FUNCTION_BLOCK FB_MockNciChannel EXTENDS FB_ComponentBase IMPLEMENTS I_NciChannel_GCode
VAR_INPUT
    MockIsGrouped      : BOOL;
    MockIsProgramLoaded: BOOL;
    MockIsReady        : BOOL;
    MockIsMoving       : BOOL;
    MockChannelError   : BOOL;
    MockChannelErrorId : UDINT;
END_VAR
VAR_OUTPUT
    BuildGroupCallCount : INT;
    LoadProgramCallCount: INT;
    StartCallCount      : INT;
    StopCallCount       : INT;
    UngroupCallCount    : INT;
    ResetCallCount      : INT;
    LoadedProgramPath   : STRING(255);
END_VAR

METHOD BuildGroup
BuildGroupCallCount := BuildGroupCallCount + 1;
END_METHOD

PROPERTY ChannelError : BOOL
GET
ChannelError := MockChannelError;
END_GET
END_PROPERTY

PROPERTY ChannelErrorId : UDINT
GET
ChannelErrorId := MockChannelErrorId;
END_GET
END_PROPERTY

PROPERTY IsGrouped : BOOL
GET
IsGrouped := MockIsGrouped;
END_GET
END_PROPERTY

PROPERTY IsMoving : BOOL
GET
IsMoving := MockIsMoving;
END_GET
END_PROPERTY

PROPERTY IsProgramLoaded : BOOL
GET
IsProgramLoaded := MockIsProgramLoaded;
END_GET
END_PROPERTY

PROPERTY IsReady : BOOL
GET
IsReady := MockIsReady;
END_GET
END_PROPERTY

METHOD LoadProgram
VAR_INPUT
    sProgramPath : STRING(255);
END_VAR
LoadProgramCallCount := LoadProgramCallCount + 1;
LoadedProgramPath := sProgramPath;
END_METHOD

METHOD ResetChannel
ResetCallCount := ResetCallCount + 1;
MockChannelError := FALSE;
MockChannelErrorId := 0;
END_METHOD

METHOD Start
StartCallCount := StartCallCount + 1;
END_METHOD

METHOD Stop
StopCallCount := StopCallCount + 1;
END_METHOD

METHOD Ungroup
UngroupCallCount := UngroupCallCount + 1;
END_METHOD

END_FUNCTION_BLOCK

(* stored: Version 1.1.0.1, ProductVersion 3.1.4024.15
   POU FB_MockNciChannel: Id {c1b2c3d4-e5f6-4789-9999-000000000010}, SpecialFunc None
   Method BuildGroup: Id {a1b2c3d4-e5f6-4789-9999-000000000011}
   Property ChannelError: Id {a1b2c3d4-e5f6-4789-9999-000000000012}
   Get Get: Id {a1b2c3d4-e5f6-4789-9999-000000000013}
   Property ChannelErrorId: Id {a1b2c3d4-e5f6-4789-9999-000000000014}
   Get Get: Id {a1b2c3d4-e5f6-4789-9999-000000000015}
   Property IsGrouped: Id {a1b2c3d4-e5f6-4789-9999-000000000016}
   Get Get: Id {a1b2c3d4-e5f6-4789-9999-000000000017}
   Property IsMoving: Id {a1b2c3d4-e5f6-4789-9999-000000000018}
   Get Get: Id {a1b2c3d4-e5f6-4789-9999-000000000019}
   Property IsProgramLoaded: Id {a1b2c3d4-e5f6-4789-9999-000000000020}
   Get Get: Id {a1b2c3d4-e5f6-4789-9999-000000000021}
   Property IsReady: Id {a1b2c3d4-e5f6-4789-9999-000000000022}
   Get Get: Id {a1b2c3d4-e5f6-4789-9999-000000000023}
   Method LoadProgram: Id {a1b2c3d4-e5f6-4789-9999-000000000024}
   Method ResetChannel: Id {a1b2c3d4-e5f6-4789-9999-000000000025}
   Method Start: Id {a1b2c3d4-e5f6-4789-9999-000000000026}
   Method Stop: Id {a1b2c3d4-e5f6-4789-9999-000000000027}
   Method Ungroup: Id {a1b2c3d4-e5f6-4789-9999-000000000028} *)
